TYPE Python_Kamera_Daten_Kommando :
STRUCT
		
		Trigger				:BOOL;
		ID					:STRING(32);
		Wafer_Type			:INT; 			
		
END_STRUCT
END_TYPE

(* stored: Version 1.1.0.1, ProductVersion 3.1.4024.12
   DUT Python_Kamera_Daten_Kommando: Id {75d9ee24-972e-48b2-a9be-36ed181a7b4d} *)
